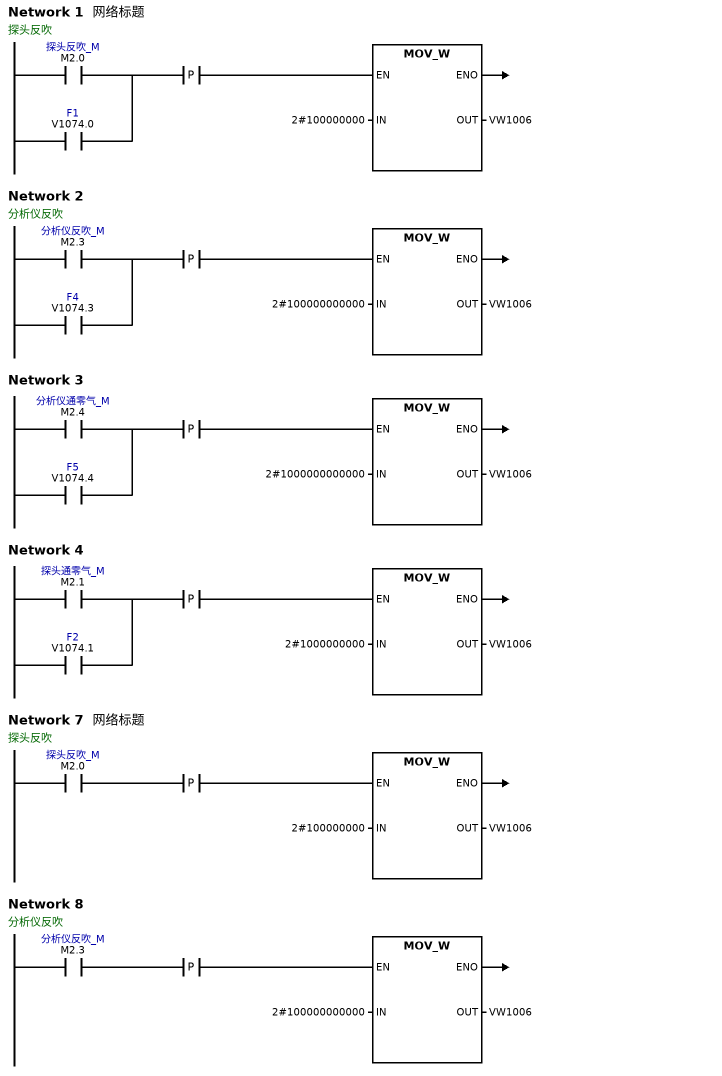
[picture p24: SBR13 networks 1-8]
Network 1 // 网络标题
// 探头反吹
LD     探头反吹_M:M2.0
O      F1:V1074.0
EU
MOVW   2#100000000, VW1006
Network 2
// 分析仪反吹
LD     分析仪反吹_M:M2.3
O      F4:V1074.3
EU
MOVW   2#100000000000, VW1006
Network 3
LD     分析仪通零气_M:M2.4
O      F5:V1074.4
EU
MOVW   2#1000000000000, VW1006
Network 4
LD     探头通零气_M:M2.1
O      F2:V1074.1
EU
MOVW   2#1000000000, VW1006
Network 7 // 网络标题
// 探头反吹
LD     探头反吹_M:M2.0
EU
MOVW   2#100000000, VW1006
Network 8
// 分析仪反吹
LD     分析仪反吹_M:M2.3
EU
MOVW   2#100000000000, VW1006
Network 10 // 网络标题
// 网络注释
END_SUBROUTINE_BLOCK

SUBROUTINE_BLOCK Manual_with_Probe_Alarm:SBR14
TITLE=子程序注释
BEGIN
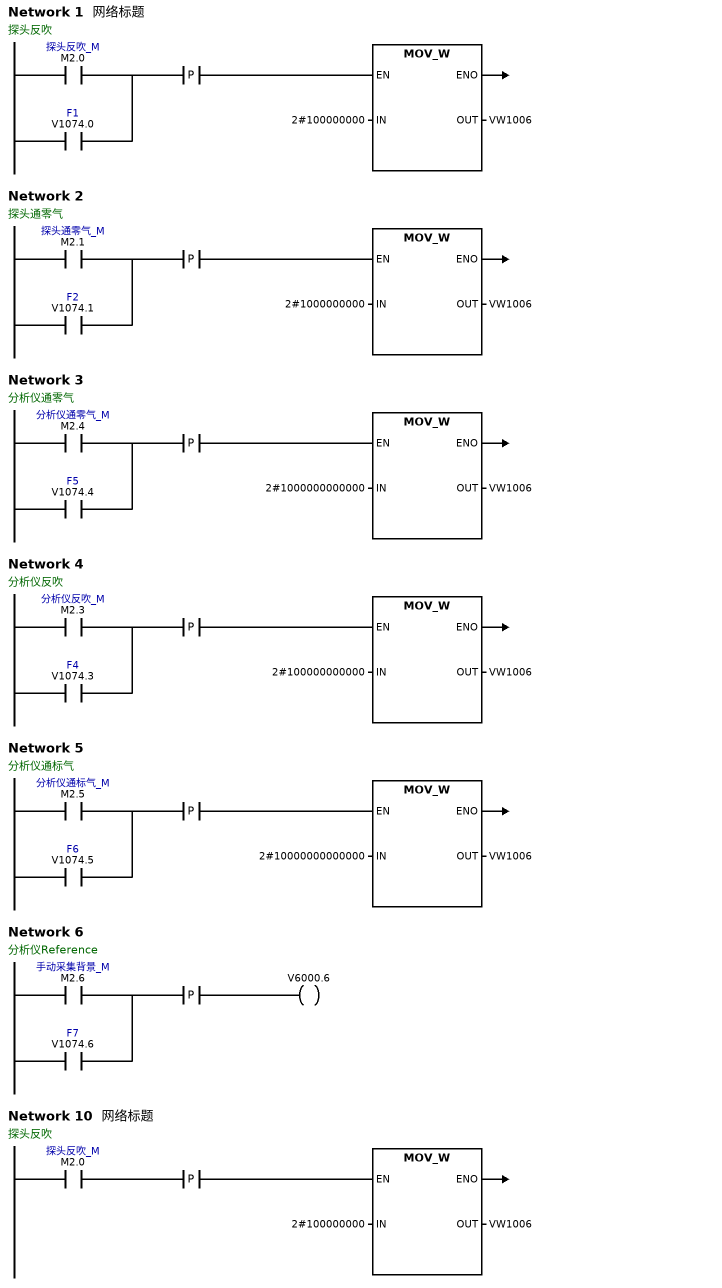
Network 1 // 网络标题
// 探头反吹
LD     探头反吹_M:M2.0
O      F1:V1074.0
EU
MOVW   2#100000000, VW1006
Network 2
// 探头通零气
LD     探头通零气_M:M2.1
O      F2:V1074.1
EU
MOVW   2#1000000000, VW1006
Network 3
// 分析仪通零气
LD     分析仪通零气_M:M2.4
O      F5:V1074.4
EU
MOVW   2#1000000000000, VW1006
Network 4
// 分析仪反吹
LD     分析仪反吹_M:M2.3
O      F4:V1074.3
EU
MOVW   2#100000000000, VW1006
Network 5
// 分析仪通标气
LD     分析仪通标气_M:M2.5
O      F6:V1074.5
EU
MOVW   2#10000000000000, VW1006
Network 6
// 分析仪Reference
LD     手动采集背景_M:M2.6
O      F7:V1074.6
EU
=      V6000.6
Network 10 // 网络标题
// 探头反吹
LD     探头反吹_M:M2.0
EU
MOVW   2#100000000, VW1006
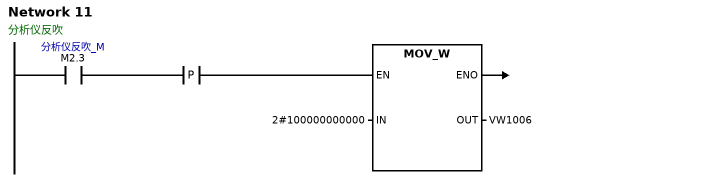
Network 11
// 分析仪反吹
LD     分析仪反吹_M:M2.3
EU
MOVW   2#100000000000, VW1006
Network 13 // 网络标题
// 网络注释
END_SUBROUTINE_BLOCK

SUBROUTINE_BLOCK AO_AI:SBR15
TITLE=
BEGIN
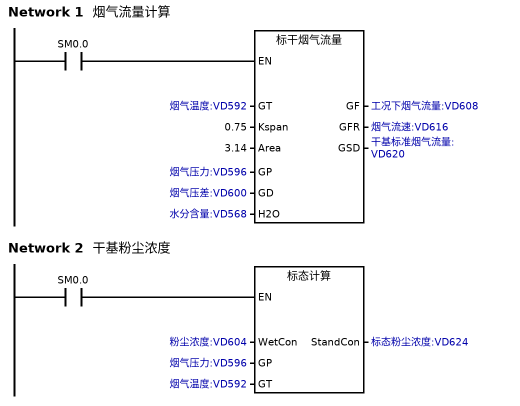
Network 1 // 烟气流量计算
LD     SM0.0
CALL   标干烟气流量:SBR20, 烟气温度:VD592, 0.75, 3.14, 烟气压力:VD596, 烟气压差:VD600, 水分含量:VD568, 工况下烟气流量:VD608, 烟气流速:VD616, 干基标准烟气流量:VD620
Network 2 // 干基粉尘浓度
LD     SM0.0
CALL   标态计算:SBR17, 粉尘浓度:VD604, 烟气压力:VD596, 烟气温度:VD592, 标态粉尘浓度:VD624
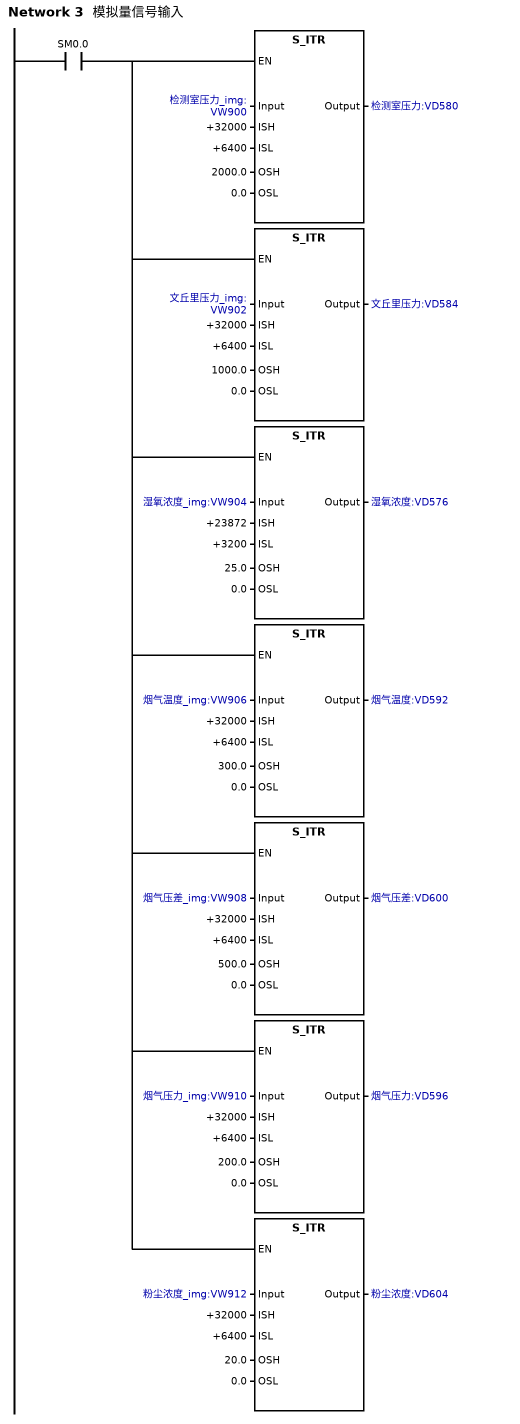
Network 3 // 模拟量信号输入
LD     SM0.0
CALL   S_ITR:SBR18, 检测室压力_img:VW900, +32000, +6400, 2000.0, 0.0, 检测室压力:VD580
CALL   S_ITR:SBR18, 文丘里压力_img:VW902, +32000, +6400, 1000.0, 0.0, 文丘里压力:VD584
CALL   S_ITR:SBR18, 湿氧浓度_img:VW904, +23872, +3200, 25.0, 0.0, 湿氧浓度:VD576
CALL   S_ITR:SBR18, 烟气温度_img:VW906, +32000, +6400, 300.0, 0.0, 烟气温度:VD592
CALL   S_ITR:SBR18, 烟气压差_img:VW908, +32000, +6400, 500.0, 0.0, 烟气压差:VD600
CALL   S_ITR:SBR18, 烟气压力_img:VW910, +32000, +6400, 200.0, 0.0, 烟气压力:VD596
CALL   S_ITR:SBR18, 粉尘浓度_img:VW912, +32000, +6400, 20.0, 0.0, 粉尘浓度:VD604
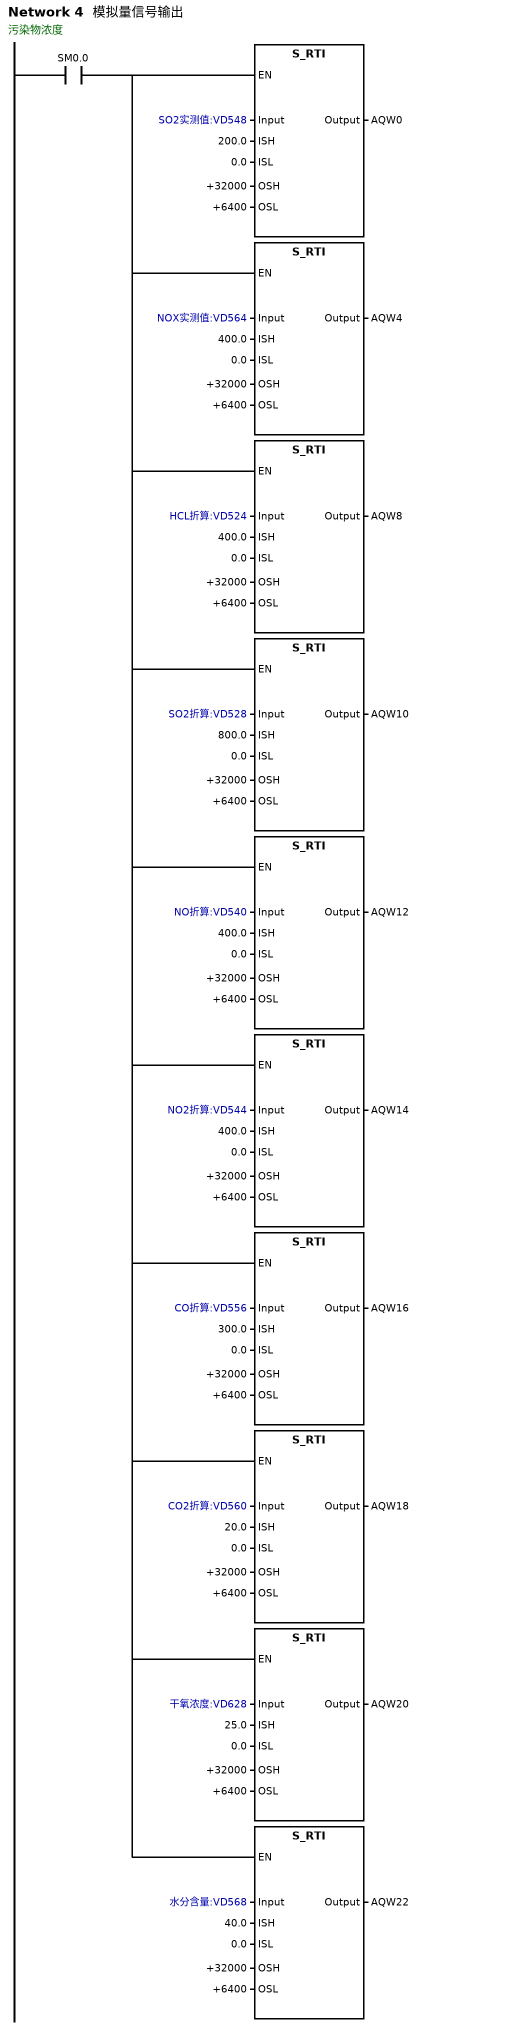
Network 4 // 模拟量信号输出
// 污染物浓度
LD     SM0.0
CALL   S_RTI:SBR19, SO2实测值:VD548, 200.0, 0.0, +32000, +6400, AQW0
CALL   S_RTI:SBR19, NOX实测值:VD564, 400.0, 0.0, +32000, +6400, AQW4
CALL   S_RTI:SBR19, HCL折算:VD524, 400.0, 0.0, +32000, +6400, AQW8
CALL   S_RTI:SBR19, SO2折算:VD528, 800.0, 0.0, +32000, +6400, AQW10
CALL   S_RTI:SBR19, NO折算:VD540, 400.0, 0.0, +32000, +6400, AQW12
CALL   S_RTI:SBR19, NO2折算:VD544, 400.0, 0.0, +32000, +6400, AQW14
CALL   S_RTI:SBR19, CO折算:VD556, 300.0, 0.0, +32000, +6400, AQW16
CALL   S_RTI:SBR19, CO2折算:VD560, 20.0, 0.0, +32000, +6400, AQW18
CALL   S_RTI:SBR19, 干氧浓度:VD628, 25.0, 0.0, +32000, +6400, AQW20
CALL   S_RTI:SBR19, 水分含量:VD568, 40.0, 0.0, +32000, +6400, AQW22
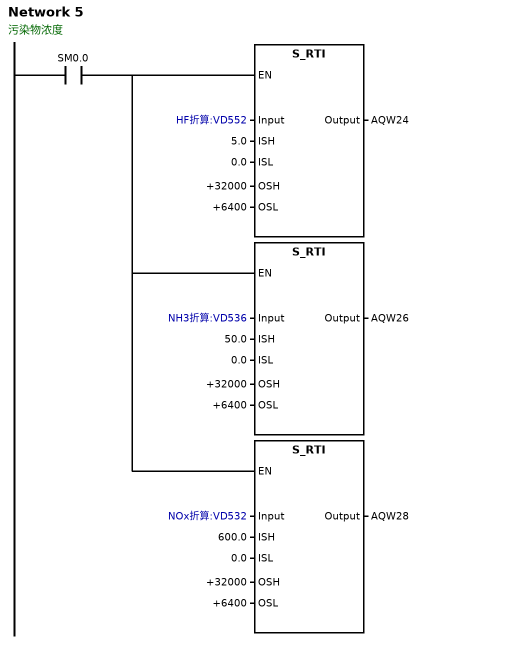
Network 5
// 污染物浓度
LD     SM0.0
CALL   S_RTI:SBR19, HF折算:VD552, 5.0, 0.0, +32000, +6400, AQW24
CALL   S_RTI:SBR19, NH3折算:VD536, 50.0, 0.0, +32000, +6400, AQW26
CALL   S_RTI:SBR19, NOx折算:VD532, 600.0, 0.0, +32000, +6400, AQW28
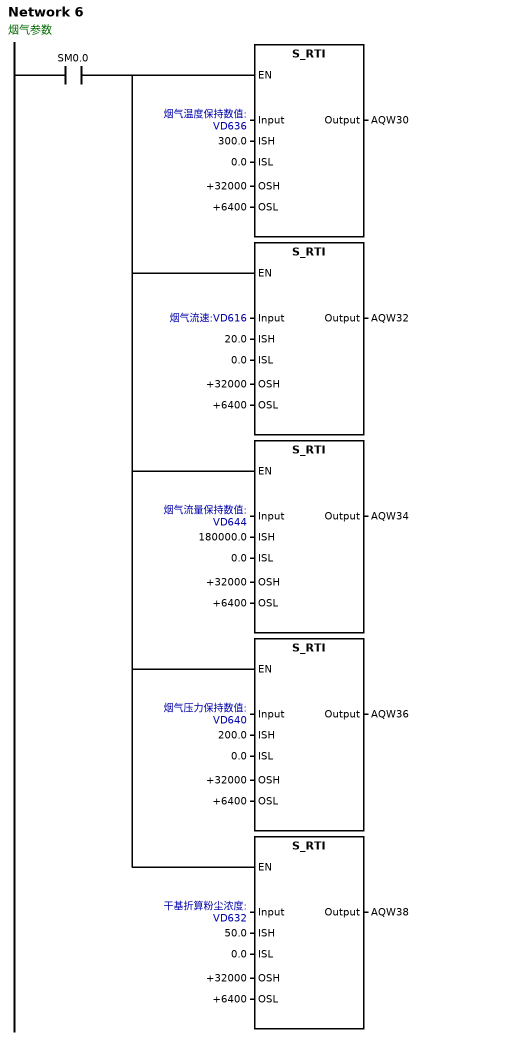
Network 6
// 烟气参数
LD     SM0.0
CALL   S_RTI:SBR19, 烟气温度保持数值:VD636, 300.0, 0.0, +32000, +6400, AQW30
CALL   S_RTI:SBR19, 烟气流速:VD616, 20.0, 0.0, +32000, +6400, AQW32
CALL   S_RTI:SBR19, 烟气流量保持数值:VD644, 180000.0, 0.0, +32000, +6400, AQW34
CALL   S_RTI:SBR19, 烟气压力保持数值:VD640, 200.0, 0.0, +32000, +6400, AQW36
CALL   S_RTI:SBR19, 干基折算粉尘浓度:VD632, 50.0, 0.0, +32000, +6400, AQW38
END_SUBROUTINE_BLOCK

SUBROUTINE_BLOCK TD400C:SBR16
TITLE=
BEGIN
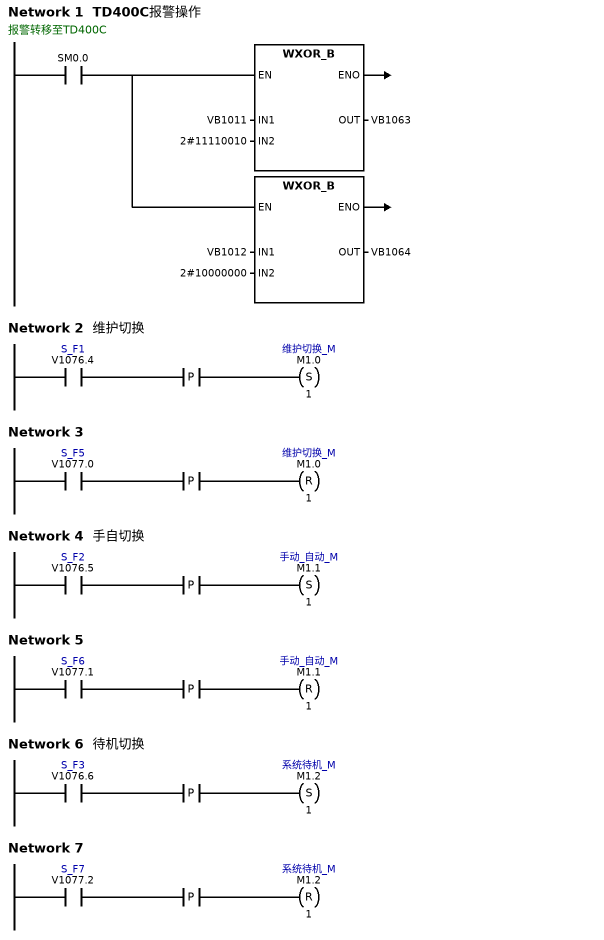
Network 1 // TD400C报警操作
// 报警转移至TD400C
LD     SM0.0
MOVB   VB1011, VB1063
XORB   2#11110010, VB1063
MOVB   VB1012, VB1064
XORB   2#10000000, VB1064
Network 2 // 维护切换
LD     S_F1:V1076.4
EU
S      维护切换_M:M1.0, 1
Network 3
LD     S_F5:V1077.0
EU
R      维护切换_M:M1.0, 1
Network 4 // 手自切换
LD     S_F2:V1076.5
EU
S      手动_自动_M:M1.1, 1
Network 5
LD     S_F6:V1077.1
EU
R      手动_自动_M:M1.1, 1
Network 6 // 待机切换
LD     S_F3:V1076.6
EU
S      系统待机_M:M1.2, 1
Network 7
LD     S_F7:V1077.2
EU
R      系统待机_M:M1.2, 1
END_SUBROUTINE_BLOCK

SUBROUTINE_BLOCK 标态计算:SBR17
TITLE=子程序注释
VAR_INPUT
WetCon:REAL;	// LD0 湿基浓度 
END_VAR
VAR_IN_OUT
GP:REAL;	// LD4 烟气压力 
GT:REAL;	// LD8 烟气温度 
END_VAR
VAR_OUTPUT
StandCon:REAL;	// LD12 标准状态浓度
END_VAR
VAR
TEMP1:REAL;	// LD16 
TEMP2:REAL;	// LD20 
TEMP3:REAL;	// LD24 
TEMP4:REAL;	// LD28 
END_VAR
BEGIN
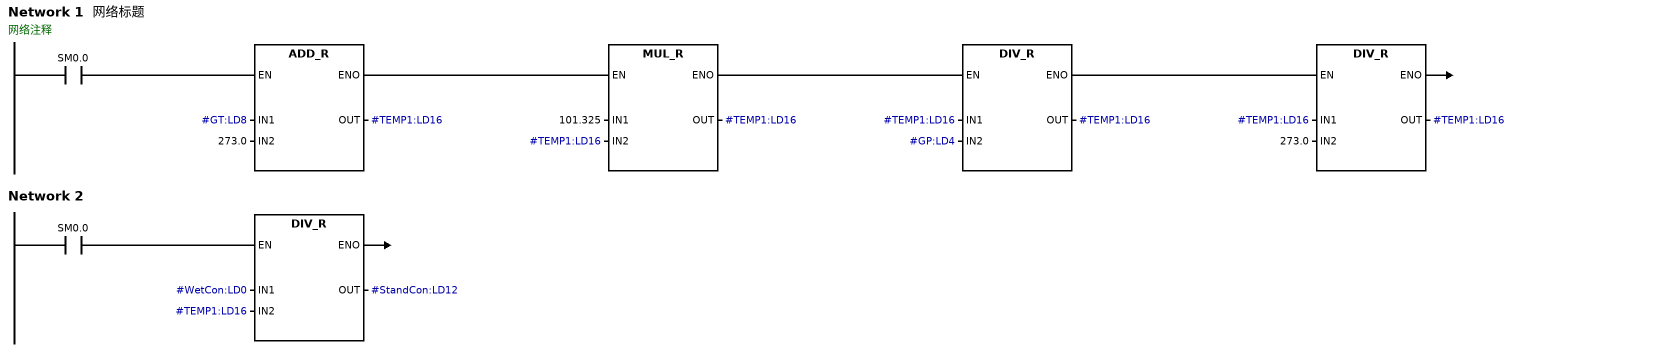
Network 1 // 网络标题
// 网络注释
LD     SM0.0
MOVR   #GT:LD8, #TEMP1:LD16
AENO
+R     273.0, #TEMP1:LD16
AENO
*R     101.325, #TEMP1:LD16
AENO
/R     #GP:LD4, #TEMP1:LD16
AENO
/R     273.0, #TEMP1:LD16
Network 2
LD     SM0.0
MOVR   #WetCon:LD0, #StandCon:LD12
/R     #TEMP1:LD16, #StandCon:LD12
END_SUBROUTINE_BLOCK

// SBR18: protected block, not included

// SBR19: protected block, not included

// SBR20: protected block, not included

SUBROUTINE_BLOCK MODBUS_Slave:SBR21
TITLE=
BEGIN
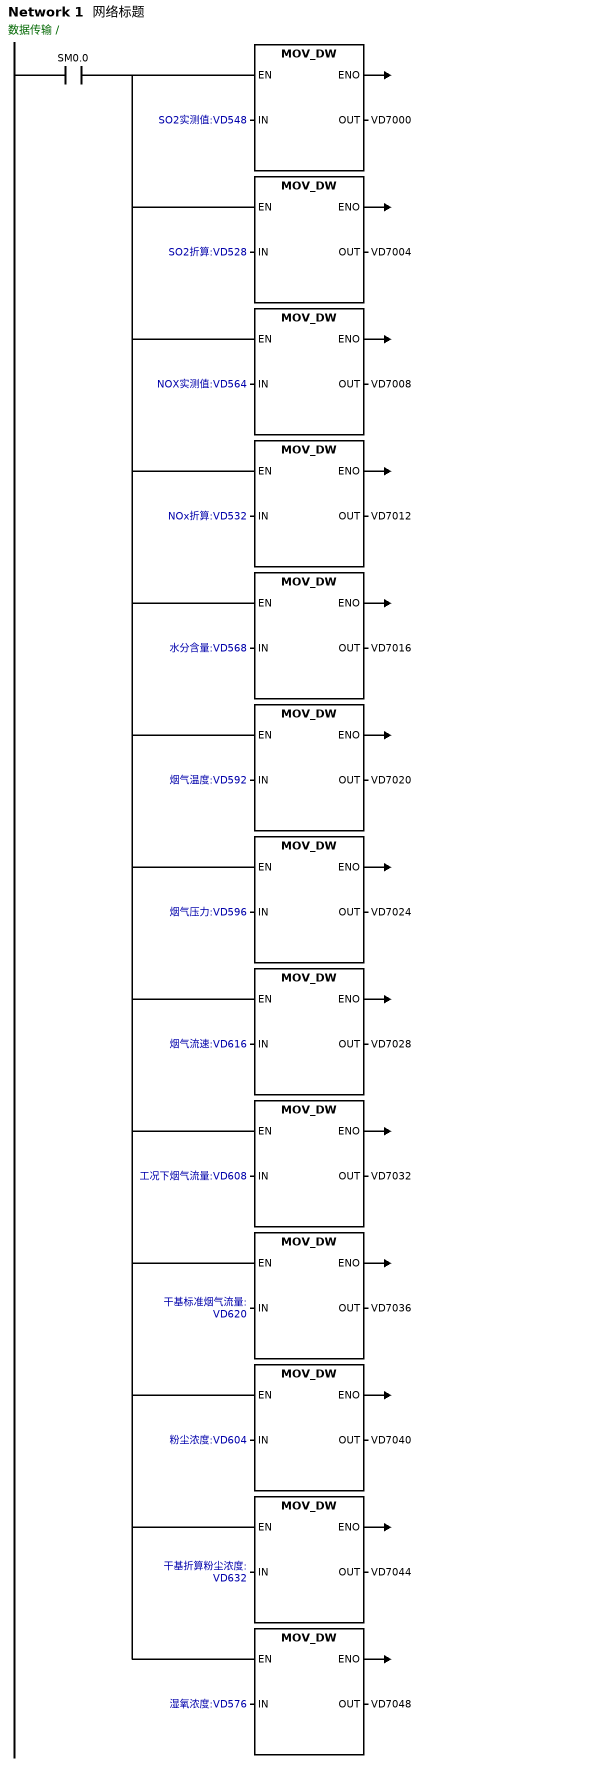
Network 1 // 网络标题
// 数据传输
// 
LD     SM0.0
MOVD   SO2实测值:VD548, VD7000
MOVD   SO2折算:VD528, VD7004
MOVD   NOX实测值:VD564, VD7008
MOVD   NOx折算:VD532, VD7012
MOVD   水分含量:VD568, VD7016
MOVD   烟气温度:VD592, VD7020
MOVD   烟气压力:VD596, VD7024
MOVD   烟气流速:VD616, VD7028
MOVD   工况下烟气流量:VD608, VD7032
MOVD   干基标准烟气流量:VD620, VD7036
MOVD   粉尘浓度:VD604, VD7040
MOVD   干基折算粉尘浓度:VD632, VD7044
MOVD   湿氧浓度:VD576, VD7048
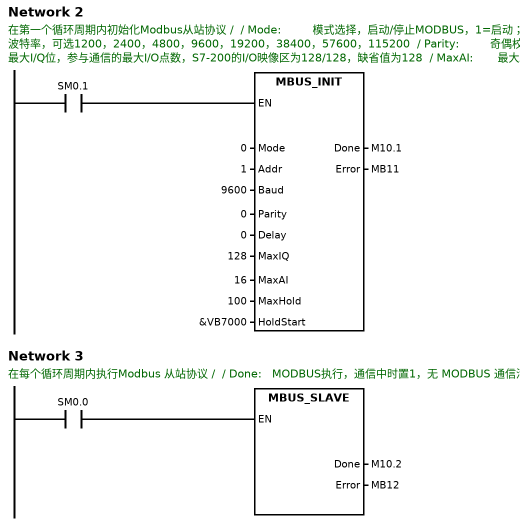
Network 2
// 在第一个循环周期内初始化Modbus从站协议
// 
// Mode:         模式选择，启动/停止MODBUS，1=启动；0=停止
// Address:     从站地址，MODBUS从站地址，取值1~247
// Baud:         波特率，可选1200，2400，4800，9600，19200，38400，57600，115200 
// Parity:         奇偶校验，0=无校验；1=奇校验；2=偶校验 
// Delay:         延时，附加字符间延时，缺省值为0 
// MaxIQ:       最大I/Q位，参与通信的最大I/O点数，S7-200的I/O映像区为128/128，缺省值为128 
// MaxAI:       最大AI字数，参与通信的最大AI通道数，可为16或32 
// MaxHold:   最大保持寄存器区，参与通信的V存储区字（VW） 
// HoldStart:   保持寄存器区起始地址，以&VBx指定（间接寻址方式） 
// 
// Done:        初始化完成标志，成功初始化后置1 
// Error:         初始化错误代码 
// 
// |
// 
// 在本例子中，设置从站地址为12
// Port0 通讯波特率为9600
// 无校验
// 可以使用的S7-200最大数字量输入输出点数为128
// 可以使用的S7-200最大模拟量输入寄存器字数为32
// 可以使用的V区寄存器地址字数为100， 起始地址为VB1000
// 
// 注意：本例子中，Modbus RTU 从站指令使用的库存储为VB0---VB779，这段寄存器地址不能再被程序中的任何指令使用，包括MBUS_INIT 和 MBUS_SLAVE 指令在内
LD     SM0.1
CALL   MBUS_INIT:SBR22, 0, 1, 9600, 0, 0, 128, 16, 100, &VB7000, M10.1, MB11
Network 3
// 在每个循环周期内执行Modbus 从站协议
// 
// Done:   MODBUS执行，通信中时置1，无 MODBUS 通信活动时为 0
// Error:    错误代码：0=无错误 
LD     SM0.0
CALL   MBUS_SLAVE:SBR23, M10.2, MB12
END_SUBROUTINE_BLOCK

// SBR22: protected block, not included

// SBR23: protected block, not included

// SBR24: protected block, not included

SUBROUTINE_BLOCK Profibus_DP:SBR25
TITLE=子程序注释
BEGIN
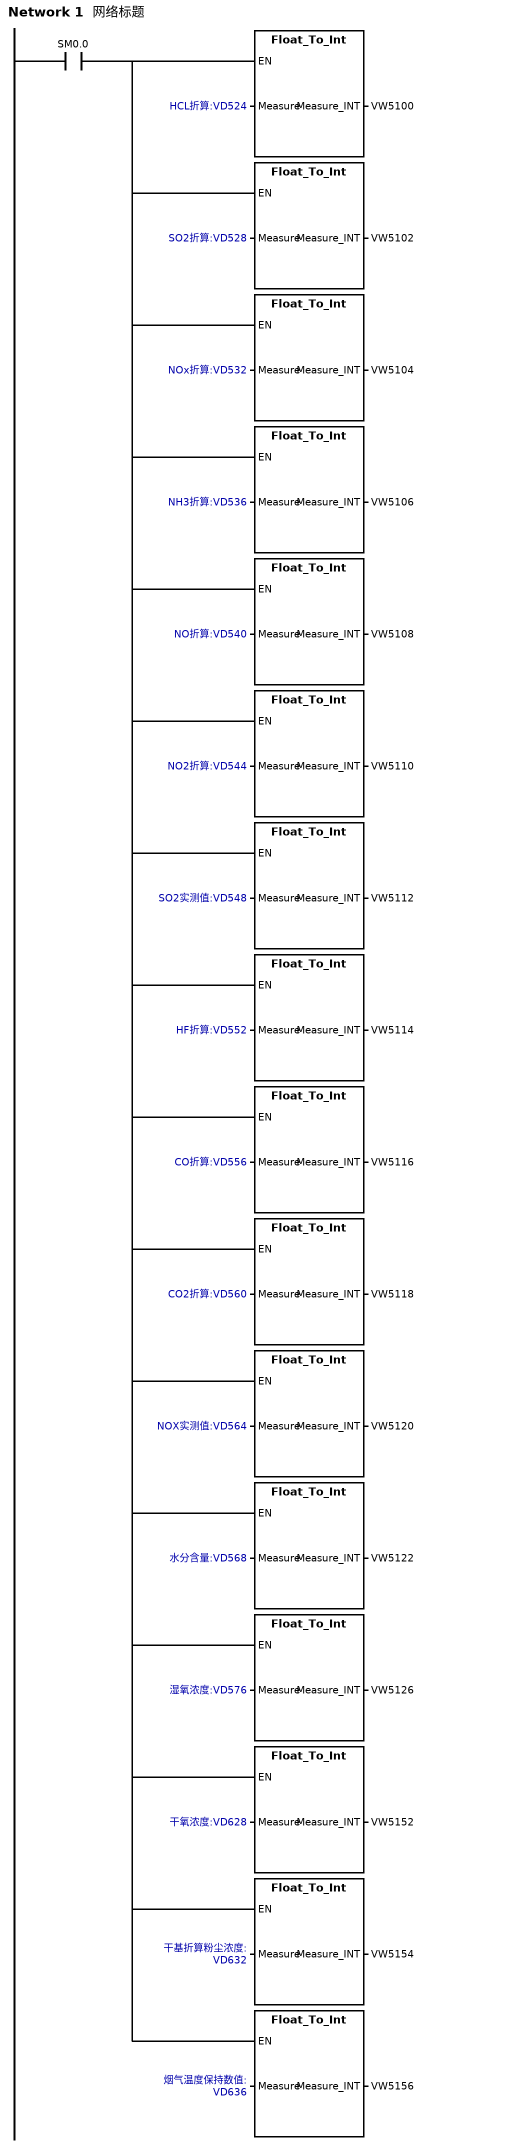
Network 1 // 网络标题
LD     SM0.0
CALL   Float_To_Int:SBR26, HCL折算:VD524, VW5100
CALL   Float_To_Int:SBR26, SO2折算:VD528, VW5102
CALL   Float_To_Int:SBR26, NOx折算:VD532, VW5104
CALL   Float_To_Int:SBR26, NH3折算:VD536, VW5106
CALL   Float_To_Int:SBR26, NO折算:VD540, VW5108
CALL   Float_To_Int:SBR26, NO2折算:VD544, VW5110
CALL   Float_To_Int:SBR26, SO2实测值:VD548, VW5112
CALL   Float_To_Int:SBR26, HF折算:VD552, VW5114
CALL   Float_To_Int:SBR26, CO折算:VD556, VW5116
CALL   Float_To_Int:SBR26, CO2折算:VD560, VW5118
CALL   Float_To_Int:SBR26, NOX实测值:VD564, VW5120
CALL   Float_To_Int:SBR26, 水分含量:VD568, VW5122
CALL   Float_To_Int:SBR26, 湿氧浓度:VD576, VW5126
CALL   Float_To_Int:SBR26, 干氧浓度:VD628, VW5152
CALL   Float_To_Int:SBR26, 干基折算粉尘浓度:VD632, VW5154
CALL   Float_To_Int:SBR26, 烟气温度保持数值:VD636, VW5156
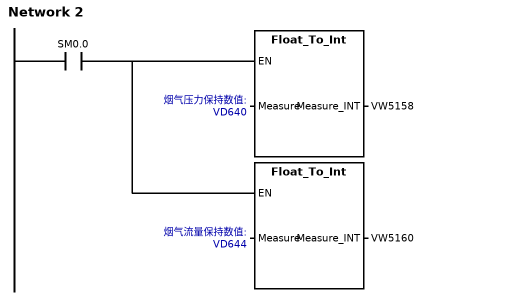
Network 2
LD     SM0.0
CALL   Float_To_Int:SBR26, 烟气压力保持数值:VD640, VW5158
CALL   Float_To_Int:SBR26, 烟气流量保持数值:VD644, VW5160
END_SUBROUTINE_BLOCK

SUBROUTINE_BLOCK Float_To_Int:SBR26
TITLE=子程序注释
VAR_INPUT
Measure:REAL;	// LD0 
END_VAR
VAR_OUTPUT
Measure_INT:WORD;	// LW4 
END_VAR
VAR
temp1:REAL;	// LD6 
temp2:DWORD;	// LD10 
END_VAR
BEGIN
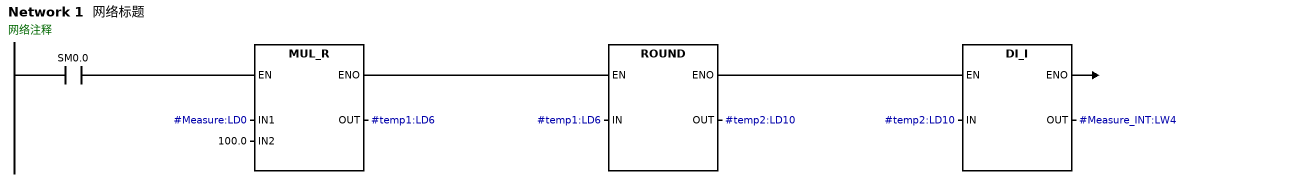
Network 1 // 网络标题
// 网络注释
LD     SM0.0
MOVR   #Measure:LD0, #temp1:LD6
AENO
*R     100.0, #temp1:LD6
AENO
ROUND  #temp1:LD6, #temp2:LD10
AENO
DTI    #temp2:LD10, #Measure_INT:LW4
END_SUBROUTINE_BLOCK

DATA_BLOCK_TAB 用户定义1
BEGIN
VD7052   3.14                //烟道截面积
VD7056   0.85                //皮托管系数
VD7060   
VD7064   200.0               //SO2量程mg/m3
VD7068   400.0               //NOx量程mg/m3
VD7072   300.0               //烟气温度量程C
VD7076   200.0               //烟气压力量程KPa
VD7080   20.0                //烟气流速量程m/s
VD7084   180000.0            //烟气流量量程m3/h
VD7088   50.0                //粉尘浓度量程
VD7092   25.0                //氧气浓度量程
VD7096   40.0                //水分含量量程
         烟气温度报警限值, 120.0
END_DATA_BLOCK_TAB

// (further data pages could not be read)
